{attribute 'qualified_only'}
VAR_GLOBAL
	mb_Input_Coils : ARRAY [0..5] OF BOOL;
	mb_Output_Coils : ARRAY [0..5] OF BOOL;
END_VAR

(* stored: Version 1.1.0.1, ProductVersion 3.1.4024.12
   GVL GVL: Id {e894af3d-25ee-4d9d-a925-7088cda0f3a6} *)
